// TIA Portal V17 export
// export: Created 2024-09-02T12:50:09.0439099Z, ExportSetting WithDefaults, DisplayName Totally Integrated Automation Portal, DisplayVersion V17, DisplayName TIA Portal Openness, DisplayVersion V17, DisplayName TIA Portal Version Control Interface, DisplayVersion V17, DisplayName STEP 7 Professional, DisplayVersion V17, DisplayName STEP 7 Safety, DisplayVersion V17, DisplayName WinCC Professional, DisplayVersion V17
FUNCTION_BLOCK "GraFB2_FG02_Station_OP70"   // FB1382, GRAPH
VERSION : 0.1
// stored: AcknowledgeErrorsRequired false, AutoNumber false, GraphVersion 4.0, InitialValuesAcquisition true, IsIECCheckEnabled false, LanguageInNetworks LAD, LockOperatingMode false, PermanentILProcessingInMANMode true, SetENOAutomatically false, SkipSteps false, UDAEnableTagReadback false, WithAlarmHandling true
   // inherited from GRAPH_BASE
   VAR
      OFF_SQ_BASE : Bool;
   END_VAR
   VAR_INPUT
      OFF_SQ { ExternalWritable := 'False'} : Bool := false;
      INIT_SQ { ExternalWritable := 'False'} : Bool := false;
      ACK_EF { ExternalWritable := 'False'} : Bool := false;
      S_PREV { ExternalWritable := 'False'} : Bool := false;
      S_NEXT { ExternalWritable := 'False'} : Bool := false;
      SW_AUTO { ExternalWritable := 'False'} : Bool := false;
      SW_TAP { ExternalWritable := 'False'} : Bool := false;
      SW_TOP { ExternalWritable := 'False'} : Bool := false;
      SW_MAN { ExternalWritable := 'False'} : Bool := false;
      S_SEL { ExternalWritable := 'False'} : Int := 0;
      S_ON { ExternalWritable := 'False'} : Bool := false;
      S_OFF { ExternalWritable := 'False'} : Bool := false;
      T_PUSH { ExternalWritable := 'False'} : Bool := false;
   END_VAR
   VAR_OUTPUT
      S_NO { ExternalWritable := 'False'} : Int := 0;
      S_MORE { ExternalWritable := 'False'} : Bool := false;
      S_ACTIVE { ExternalWritable := 'False'} : Bool := false;
      ERR_FLT { ExternalWritable := 'False'} : Bool := false;
      AUTO_ON { ExternalWritable := 'False'} : Bool := false;
      TAP_ON { ExternalWritable := 'False'} : Bool := false;
      TOP_ON { ExternalWritable := 'False'} : Bool := false;
      MAN_ON { ExternalWritable := 'False'} : Bool := false;
   END_VAR
   VAR
      extBlock { S7_SetPoint := 'True'} : "LTLL_ManualGraphExt";
   END_VAR
BEGIN
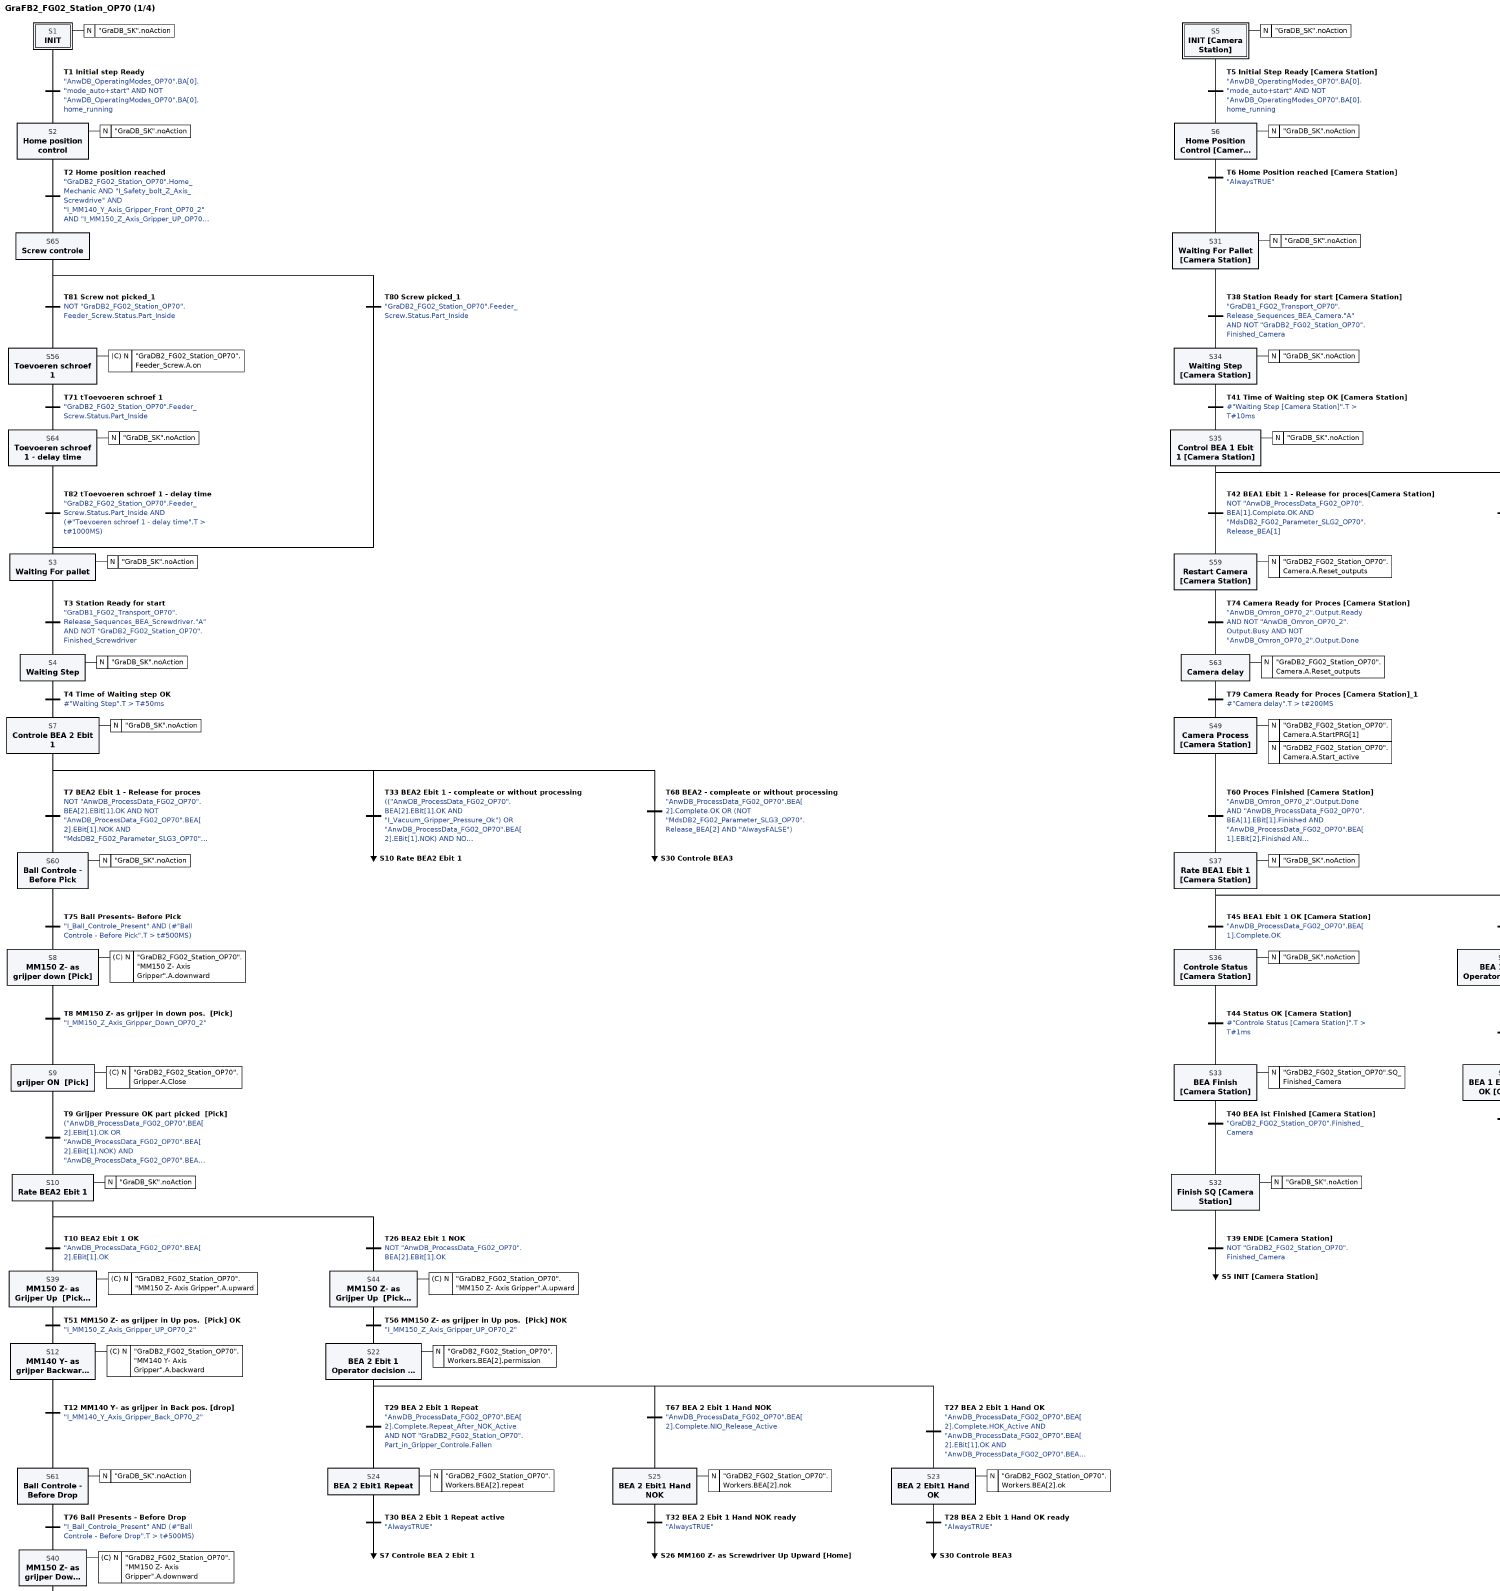
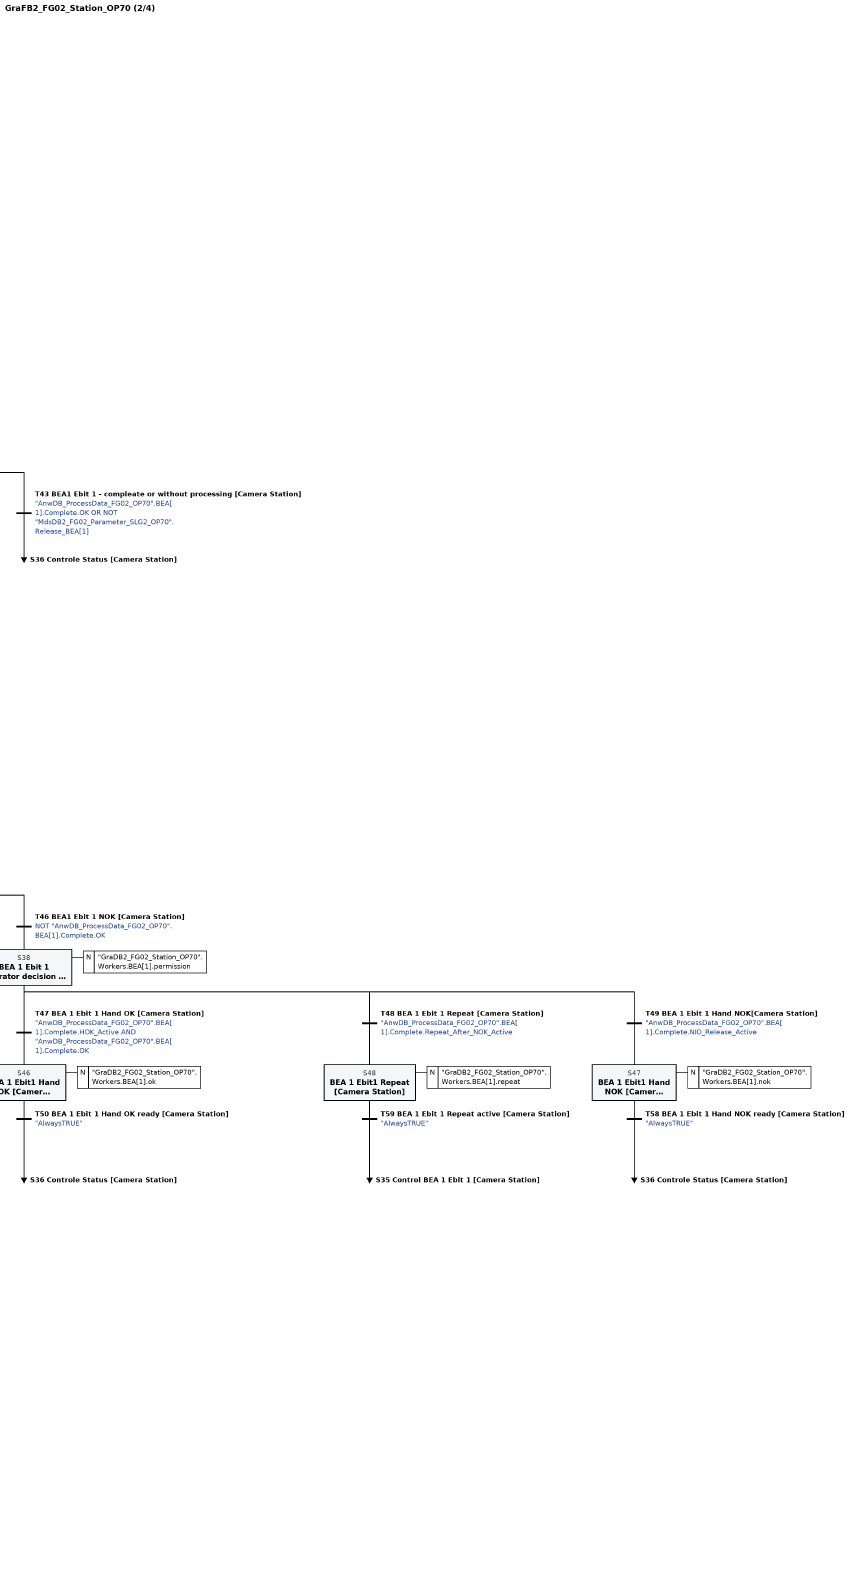
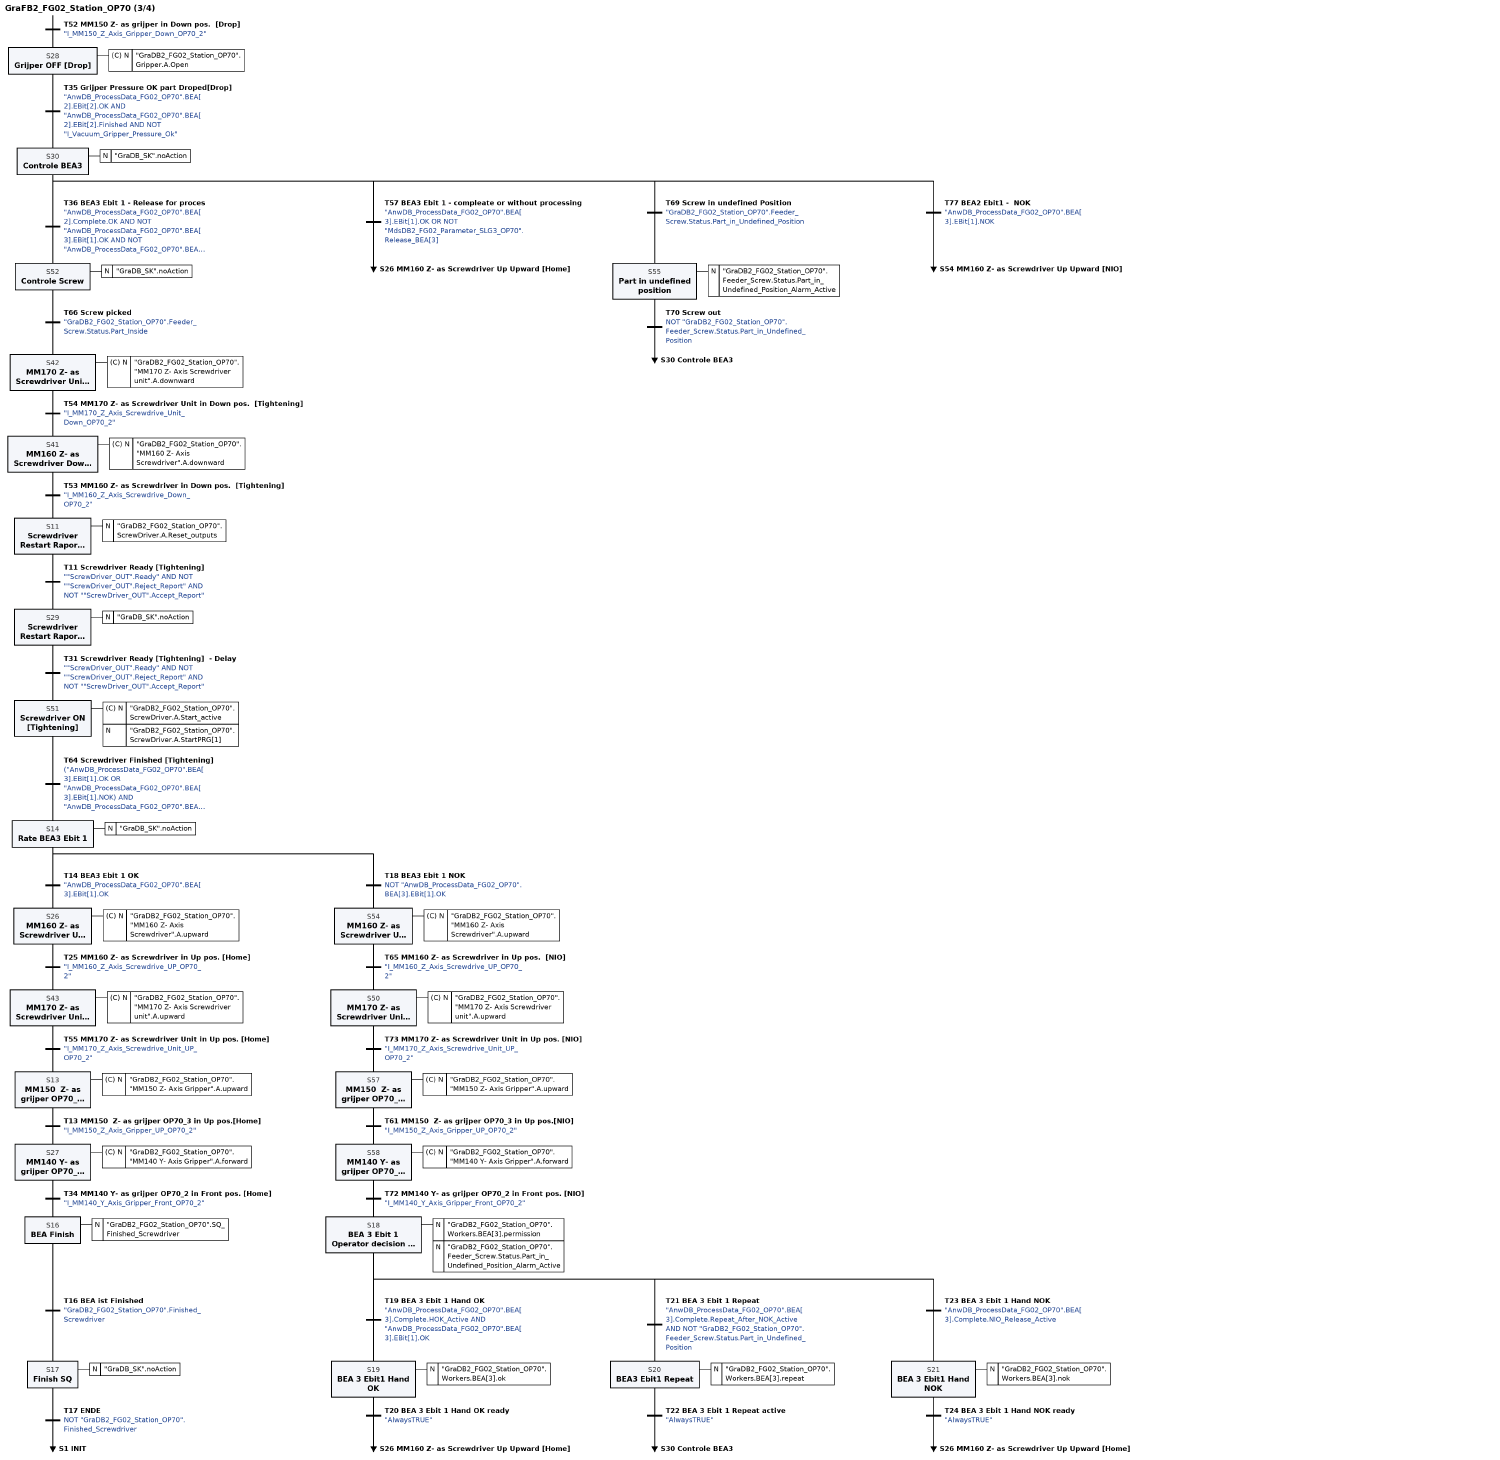
   // permanent pre-instructions
   NETWORK 1
   TITLE = HMI Lite Pass on data
      #extBlock.input := "LTLL_ManualGraphControl_OP70".screen[0].input;
   NETWORK 2
   TITLE = Instance DB Name query and pass on
      GetInstanceName(size := 0, OUT => #extBlock.input.instanceName);
   NETWORK 3
   TITLE = SK Mode
      "SysFC_SQ_Mode"(iFKT := 0, iTmsHalt := false, ioMOP := #RT_DATA.MOP);

   // sequencer 1: Station cycle Screwdriver
   // sample
   INITIAL_STEP INIT:   // S1, max time T#10S, warning time T#7S: Step commentary
      interlock C := (none);   // initial step
      supervision V := (none);   // initial step
              N    "GraDB_SK".noAction
   END_STEP
   TRANSITION "Initial step Ready" FROM INIT TO "Home position control"   // T1
      := "AnwDB_OperatingModes_OP70".BA[0]."mode_auto+start" AND NOT "AnwDB_OperatingModes_OP70".BA[0].home_running;
   END_TRANSITION
   STEP "Home position control":   // S2, max time T#10S, warning time T#7S
      supervision V := NOT #"Home position reached".TT AND (#"Home position control".U > T#1S);
      // Station
              N    "GraDB_SK".noAction
   END_STEP
   TRANSITION "Home position reached" FROM "Home position control" TO "Screw controle"   // T2
      := "GraDB2_FG02_Station_OP70".Home_Mechanic AND "I_Safety_bolt_Z_Axis_Screwdrive" AND "I_MM140_Y_Axis_Gripper_Front_OP70_2" AND "I_MM150_Z_Axis_Gripper_UP_OP70_2" AND "I_MM160_Z_Axis_Screwdrive_UP_OP70_2" AND "I_MM170_Z_Axis_Screwdrive_Unit_UP_OP70_2";
   END_TRANSITION
   STEP "Waiting For pallet":   // S3, max time T#10S, warning time T#7S
              N    "GraDB_SK".noAction
   END_STEP
   TRANSITION "Station Ready for start" FROM "Waiting For pallet" TO "Waiting Step"   // T3
      := "GraDB1_FG02_Transport_OP70".Release_Sequences_BEA_Screwdriver."A" AND NOT "GraDB2_FG02_Station_OP70".Finished_Screwdriver;
   END_TRANSITION
   STEP "Finish SQ":   // S17, max time T#10S, warning time T#7S
              N    "GraDB_SK".noAction
   END_STEP
   TRANSITION ENDE FROM "Finish SQ" TO INIT   // T17, jump
      := NOT "GraDB2_FG02_Station_OP70".Finished_Screwdriver;
   END_TRANSITION
   STEP "BEA Finish":   // S16, max time T#10S, warning time T#7S
      supervision V := NOT #"BEA ist Finished".TT AND (#"BEA Finish".U > T#1000ms);
              N    "GraDB2_FG02_Station_OP70".SQ_Finished_Screwdriver
   END_STEP
   TRANSITION "BEA ist Finished" FROM "BEA Finish" TO "Finish SQ"   // T16
      := "GraDB2_FG02_Station_OP70".Finished_Screwdriver;
   END_TRANSITION
   STEP "Waiting Step":   // S4, max time T#10S, warning time T#7S
      supervision V := NOT #"Time of Waiting step OK".TT AND (#"Waiting Step".U > t#1S);
              N    "GraDB_SK".noAction
   END_STEP
   TRANSITION "Time of Waiting step OK" FROM "Waiting Step" TO "Controle BEA 2 Ebit 1"   // T4
      := #"Waiting Step".T > T#50ms;
   END_TRANSITION
   STEP "Controle BEA 2 Ebit 1":   // S7, max time T#10S, warning time T#7S
      supervision V := NOT #"BEA2 Ebit 1 - Release for proces".TT AND (#"Controle BEA 2 Ebit 1".U > t#1s);
              N    "GraDB_SK".noAction
   END_STEP
   TRANSITION "BEA2 Ebit 1 - Release for proces" FROM "Controle BEA 2 Ebit 1" TO "Ball Controle - Before Pick"   // T7
      := NOT "AnwDB_ProcessData_FG02_OP70".BEA[2].EBit[1].OK AND NOT "AnwDB_ProcessData_FG02_OP70".BEA[2].EBit[1].NOK AND "MdsDB2_FG02_Parameter_SLG3_OP70".Release_BEA[2];
   END_TRANSITION
   TRANSITION "BEA2 Ebit 1 - compleate or without processing" FROM "Controle BEA 2 Ebit 1" TO "Rate BEA2 Ebit 1"   // T33, jump
      := (("AnwDB_ProcessData_FG02_OP70".BEA[2].EBit[1].OK AND "I_Vacuum_Gripper_Pressure_Ok") OR "AnwDB_ProcessData_FG02_OP70".BEA[2].EBit[1].NOK) AND NOT "AnwDB_ProcessData_FG02_OP70".BEA[2].EBit[2].OK;
   END_TRANSITION
   TRANSITION "BEA2 - compleate or without processing" FROM "Controle BEA 2 Ebit 1" TO "Controle BEA3"   // T68, jump
      := "AnwDB_ProcessData_FG02_OP70".BEA[2].Complete.OK OR (NOT "MdsDB2_FG02_Parameter_SLG3_OP70".Release_BEA[2] AND "AlwaysFALSE");
   END_TRANSITION
   STEP "Rate BEA2 Ebit 1":   // S10, max time T#10S, warning time T#7S: When operator access is required
      supervision V := NOT #"BEA2 Ebit 1 OK".TT AND (#"Rate BEA2 Ebit 1".U > t#1s);
              N    "GraDB_SK".noAction
   END_STEP
   TRANSITION "BEA2 Ebit 1 OK" FROM "Rate BEA2 Ebit 1" TO "MM150 Z- as Grijper Up  [Pick] OK"   // T10
      := "AnwDB_ProcessData_FG02_OP70".BEA[2].EBit[1].OK;
   END_TRANSITION
   TRANSITION "BEA2 Ebit 1 NOK" FROM "Rate BEA2 Ebit 1" TO "MM150 Z- as Grijper Up  [Pick] NOK"   // T26
      := NOT "AnwDB_ProcessData_FG02_OP70".BEA[2].EBit[1].OK;
   END_TRANSITION
   STEP "BEA 2 Ebit 1 Operator decision - After NOK":   // S22, max time T#10S, warning time T#7S
      interlock C := "GraDB1_FG02_Transport_OP70".Release_Sequences_BEA_Screwdriver."A";
              N    "GraDB2_FG02_Station_OP70".Workers.BEA[2].permission
   END_STEP
   TRANSITION "BEA 2 Ebit 1 Repeat" FROM "BEA 2 Ebit 1 Operator decision - After NOK" TO "BEA 2 Ebit1 Repeat"   // T29
      := "AnwDB_ProcessData_FG02_OP70".BEA[2].Complete.Repeat_After_NOK_Active AND NOT "GraDB2_FG02_Station_OP70".Part_in_Gripper_Controle.Fallen;
   END_TRANSITION
   TRANSITION "BEA 2 Ebit 1 Hand NOK" FROM "BEA 2 Ebit 1 Operator decision - After NOK" TO "BEA 2 Ebit1 Hand NOK"   // T67
      := "AnwDB_ProcessData_FG02_OP70".BEA[2].Complete.NIO_Release_Active;
   END_TRANSITION
   TRANSITION "BEA 2 Ebit 1 Hand OK" FROM "BEA 2 Ebit 1 Operator decision - After NOK" TO "BEA 2 Ebit1 Hand OK"   // T27
      := "AnwDB_ProcessData_FG02_OP70".BEA[2].Complete.HOK_Active AND "AnwDB_ProcessData_FG02_OP70".BEA[2].EBit[1].OK AND "AnwDB_ProcessData_FG02_OP70".BEA[2].EBit[2].OK AND NOT "GraDB2_FG02_Station_OP70".Part_in_Gripper_Controle.Fallen;
   END_TRANSITION
   STEP "BEA 2 Ebit1 Hand NOK":   // S25, max time T#10S, warning time T#7S
              N    "GraDB2_FG02_Station_OP70".Workers.BEA[2].nok
   END_STEP
   TRANSITION "BEA 2 Ebit 1 Hand NOK ready" FROM "BEA 2 Ebit1 Hand NOK" TO "MM160 Z- as Screwdriver Up Upward [Home]"   // T32, jump
      := "AlwaysTRUE";
   END_TRANSITION
   STEP "BEA 2 Ebit1 Repeat":   // S24, max time T#10S, warning time T#7S
              N    "GraDB2_FG02_Station_OP70".Workers.BEA[2].repeat
   END_STEP
   TRANSITION "BEA 2 Ebit 1 Repeat active" FROM "BEA 2 Ebit1 Repeat" TO "Controle BEA 2 Ebit 1"   // T30, jump
      := "AlwaysTRUE";
   END_TRANSITION
   STEP "MM150 Z- as Grijper Up  [Pick] OK":   // S39, max time T#10S, warning time T#7S
      interlock C := "I_MM140_Y_Axis_Gripper_Front_OP70_2" AND "I_Vacuum_Gripper_Pressure_Ok" AND NOT "AnwDB_ProcessData_FG02_OP70".BEA[2].EBit[1].NOK;
      supervision V := NOT #"MM150 Z- as grijper in Up pos.  [Pick] OK".TT AND (#"MM150 Z- as Grijper Up  [Pick] OK".U > t#1S);
      (C)     N    "GraDB2_FG02_Station_OP70"."MM150 Z- Axis Gripper".A.upward
   END_STEP
   TRANSITION "MM150 Z- as grijper in Up pos.  [Pick] OK" FROM "MM150 Z- as Grijper Up  [Pick] OK" TO "MM140 Y- as grijper Backward [drop]"   // T51
      := "I_MM150_Z_Axis_Gripper_UP_OP70_2";
   END_TRANSITION
   STEP "MM150 Z- as grijper down [Pick]":   // S8, max time T#10S, warning time T#7S
      interlock C := "I_MM70/71_index_Screwdriver_UP_OP70_2" AND "I_MM140_Y_Axis_Gripper_Front_OP70_2" AND NOT "I_Vacuum_Gripper_Pressure_Ok" AND NOT "AnwDB_ProcessData_FG02_OP70".BEA[2].EBit[1].OK;
      supervision V := NOT #"MM150 Z- as grijper in down pos.  [Pick]".TT AND (#"MM150 Z- as grijper down [Pick]".U > t#1S);
      (C)     N    "GraDB2_FG02_Station_OP70"."MM150 Z- Axis Gripper".A.downward
   END_STEP
   TRANSITION "MM150 Z- as grijper in down pos.  [Pick]" FROM "MM150 Z- as grijper down [Pick]" TO "grijper ON  [Pick]"   // T8
      := "I_MM150_Z_Axis_Gripper_Down_OP70_2";
   END_TRANSITION
   STEP "grijper ON  [Pick]":   // S9, max time T#10S, warning time T#7S
      interlock C := "I_MM70/71_index_Screwdriver_UP_OP70_2" AND "I_MM140_Y_Axis_Gripper_Front_OP70_2" AND "I_MM150_Z_Axis_Gripper_Down_OP70_2";
      supervision V := NOT #"Grijper Pressure OK part picked  [Pick]".TT AND (#"grijper ON  [Pick]".U > t#1S);
      (C)     N    "GraDB2_FG02_Station_OP70".Gripper.A.Close
   END_STEP
   TRANSITION "Grijper Pressure OK part picked  [Pick]" FROM "grijper ON  [Pick]" TO "Rate BEA2 Ebit 1"   // T9
      := ("AnwDB_ProcessData_FG02_OP70".BEA[2].EBit[1].OK OR "AnwDB_ProcessData_FG02_OP70".BEA[2].EBit[1].NOK) AND "AnwDB_ProcessData_FG02_OP70".BEA[2].EBit[1].Finished;
   END_TRANSITION
   STEP "Rate BEA3 Ebit 1":   // S14, max time T#10S, warning time T#7S: When operator access is required
      supervision V := NOT #"BEA3 Ebit 1 OK".TT AND (#"Rate BEA3 Ebit 1".U > t#1s);
              N    "GraDB_SK".noAction
   END_STEP
   TRANSITION "BEA3 Ebit 1 OK" FROM "Rate BEA3 Ebit 1" TO "MM160 Z- as Screwdriver Up Upward [Home]"   // T14
      := "AnwDB_ProcessData_FG02_OP70".BEA[3].EBit[1].OK;
   END_TRANSITION
   TRANSITION "BEA3 Ebit 1 NOK" FROM "Rate BEA3 Ebit 1" TO "MM160 Z- as Screwdriver Up Upward [NIO]"   // T18
      := NOT "AnwDB_ProcessData_FG02_OP70".BEA[3].EBit[1].OK;
   END_TRANSITION
   STEP "BEA 3 Ebit 1 Operator decision - After NOK":   // S18, max time T#10S, warning time T#7S
      interlock C := "GraDB1_FG02_Transport_OP70".Release_Sequences_BEA_Screwdriver."A";
              N    "GraDB2_FG02_Station_OP70".Workers.BEA[3].permission
              N    "GraDB2_FG02_Station_OP70".Feeder_Screw.Status.Part_in_Undefined_Position_Alarm_Active
   END_STEP
   TRANSITION "BEA 3 Ebit 1 Hand OK" FROM "BEA 3 Ebit 1 Operator decision - After NOK" TO "BEA 3 Ebit1 Hand OK"   // T19
      := "AnwDB_ProcessData_FG02_OP70".BEA[3].Complete.HOK_Active AND "AnwDB_ProcessData_FG02_OP70".BEA[3].EBit[1].OK;
   END_TRANSITION
   TRANSITION "BEA 3 Ebit 1 Repeat" FROM "BEA 3 Ebit 1 Operator decision - After NOK" TO "BEA3 Ebit1 Repeat"   // T21
      := "AnwDB_ProcessData_FG02_OP70".BEA[3].Complete.Repeat_After_NOK_Active AND NOT "GraDB2_FG02_Station_OP70".Feeder_Screw.Status.Part_in_Undefined_Position;
   END_TRANSITION
   TRANSITION "BEA 3 Ebit 1 Hand NOK" FROM "BEA 3 Ebit 1 Operator decision - After NOK" TO "BEA 3 Ebit1 Hand NOK"   // T23
      := "AnwDB_ProcessData_FG02_OP70".BEA[3].Complete.NIO_Release_Active;
   END_TRANSITION
   STEP "BEA 3 Ebit1 Hand OK":   // S19, max time T#10S, warning time T#7S
              N    "GraDB2_FG02_Station_OP70".Workers.BEA[3].ok
   END_STEP
   TRANSITION "BEA 3 Ebit 1 Hand OK ready" FROM "BEA 3 Ebit1 Hand OK" TO "MM160 Z- as Screwdriver Up Upward [Home]"   // T20, jump
      := "AlwaysTRUE";
   END_TRANSITION
   STEP "BEA 3 Ebit1 Hand NOK":   // S21, max time T#10S, warning time T#7S
              N    "GraDB2_FG02_Station_OP70".Workers.BEA[3].nok
   END_STEP
   TRANSITION "BEA 3 Ebit 1 Hand NOK ready" FROM "BEA 3 Ebit1 Hand NOK" TO "MM160 Z- as Screwdriver Up Upward [Home]"   // T24, jump
      := "AlwaysTRUE";
   END_TRANSITION
   STEP "BEA3 Ebit1 Repeat":   // S20, max time T#10S, warning time T#7S
              N    "GraDB2_FG02_Station_OP70".Workers.BEA[3].repeat
   END_STEP
   TRANSITION "BEA 3 Ebit 1 Repeat active" FROM "BEA3 Ebit1 Repeat" TO "Controle BEA3"   // T22, jump
      := "AlwaysTRUE";
   END_TRANSITION
   STEP "MM150 Z- as grijper Down [Drop]":   // S40, max time T#10S, warning time T#7S
      interlock C := "I_MM70/71_index_Screwdriver_UP_OP70_2" AND "I_MM140_Y_Axis_Gripper_Back_OP70_2" AND "I_Vacuum_Gripper_Pressure_Ok" AND "AnwDB_ProcessData_FG02_OP70".BEA[2].EBit[1].OK AND NOT "AnwDB_ProcessData_FG02_OP70".BEA[2].EBit[1].NOK;
      supervision V := NOT #"MM150 Z- as grijper in Down pos.  [Drop]".TT AND (#"MM150 Z- as grijper Down [Drop]".U > t#1S);
      (C)     N    "GraDB2_FG02_Station_OP70"."MM150 Z- Axis Gripper".A.downward
   END_STEP
   TRANSITION "MM150 Z- as grijper in Down pos.  [Drop]" FROM "MM150 Z- as grijper Down [Drop]" TO "Grijper OFF [Drop]"   // T52
      := "I_MM150_Z_Axis_Gripper_Down_OP70_2";
   END_TRANSITION
   STEP "Screwdriver Restart Raport [Tightening]":   // S11, max time T#10S, warning time T#7S
      interlock C := "AlwaysTRUE";
      supervision V := NOT #"Screwdriver Ready [Tightening]".TT AND (#"Screwdriver Restart Raport [Tightening]".U > t#10S);
              N    "GraDB2_FG02_Station_OP70".ScrewDriver.A.Reset_outputs
   END_STEP
   TRANSITION "Screwdriver Ready [Tightening]" FROM "Screwdriver Restart Raport [Tightening]" TO "Screwdriver Restart Raport [Tightening] - Delay"   // T11
      := ""ScrewDriver_OUT".Ready" AND NOT ""ScrewDriver_OUT".Reject_Report" AND NOT ""ScrewDriver_OUT".Accept_Report";
   END_TRANSITION
   STEP "MM160 Z- as Screwdriver Up Upward [Home]":   // S26, max time T#10S, warning time T#7S
      interlock C := "AlwaysTRUE";
      supervision V := NOT #"MM160 Z- as Screwdriver in Up pos. [Home]".TT AND (#"MM160 Z- as Screwdriver Up Upward [Home]".U > T#5S);
      (C)     N    "GraDB2_FG02_Station_OP70"."MM160 Z- Axis Screwdriver".A.upward
   END_STEP
   TRANSITION "MM160 Z- as Screwdriver in Up pos. [Home]" FROM "MM160 Z- as Screwdriver Up Upward [Home]" TO "MM170 Z- as Screwdriver Unit Up [Home]"   // T25
      := "I_MM160_Z_Axis_Screwdrive_UP_OP70_2";
   END_TRANSITION
   STEP "MM160 Z- as Screwdriver Down [Tightening]":   // S41, max time T#10S, warning time T#7S
      interlock C := "I_MM70/71_index_Screwdriver_UP_OP70_2" AND "I_MM170_Z_Axis_Screwdrive_Unit_Down_OP70_2" AND (("I_MM140_Y_Axis_Gripper_Back_OP70_2" AND "I_MM150_Z_Axis_Gripper_Down_OP70_2") OR ("I_MM140_Y_Axis_Gripper_Front_OP70_2" AND "I_MM150_Z_Axis_Gripper_UP_OP70_2")) AND "AnwDB_ProcessData_FG02_OP70".BEA[2].Complete.OK;
      supervision V := NOT #"MM160 Z- as Screwdriver in Down pos.  [Tightening]".TT AND (#"MM160 Z- as Screwdriver Down [Tightening]".U > t#1S);
      (C)     N    "GraDB2_FG02_Station_OP70"."MM160 Z- Axis Screwdriver".A.downward
   END_STEP
   TRANSITION "MM160 Z- as Screwdriver in Down pos.  [Tightening]" FROM "MM160 Z- as Screwdriver Down [Tightening]" TO "Screwdriver Restart Raport [Tightening]"   // T53
      := "I_MM160_Z_Axis_Screwdrive_Down_OP70_2";
   END_TRANSITION
   STEP "MM170 Z- as Screwdriver Unit Down [Tightening]":   // S42, max time T#10S, warning time T#7S
      interlock C := "I_MM70/71_index_Screwdriver_UP_OP70_2" AND "I_MM160_Z_Axis_Screwdrive_UP_OP70_2" AND (("I_MM140_Y_Axis_Gripper_Back_OP70_2" AND "I_MM150_Z_Axis_Gripper_Down_OP70_2") OR ("I_MM140_Y_Axis_Gripper_Front_OP70_2" AND "I_MM150_Z_Axis_Gripper_UP_OP70_2")) AND "I_Safety_bolt_Z_Axis_Screwdrive" AND "AnwDB_ProcessData_FG02_OP70".BEA[2].Complete.OK;
      supervision V := NOT #"MM170 Z- as Screwdriver Unit in Down pos.  [Tightening]".TT AND (#"MM170 Z- as Screwdriver Unit Down [Tightening]".U > t#1S);
      (C)     N    "GraDB2_FG02_Station_OP70"."MM170 Z- Axis Screwdriver unit".A.downward
   END_STEP
   TRANSITION "MM170 Z- as Screwdriver Unit in Down pos.  [Tightening]" FROM "MM170 Z- as Screwdriver Unit Down [Tightening]" TO "MM160 Z- as Screwdriver Down [Tightening]"   // T54
      := "I_MM170_Z_Axis_Screwdrive_Unit_Down_OP70_2";
   END_TRANSITION
   STEP "MM170 Z- as Screwdriver Unit Up [Home]":   // S43, max time T#10S, warning time T#7S
      interlock C := "I_MM160_Z_Axis_Screwdrive_UP_OP70_2" AND (("I_MM140_Y_Axis_Gripper_Back_OP70_2" AND "I_MM150_Z_Axis_Gripper_Down_OP70_2") OR ("I_MM140_Y_Axis_Gripper_Front_OP70_2" AND "I_MM150_Z_Axis_Gripper_UP_OP70_2")) AND "I_Safety_bolt_Z_Axis_Screwdrive";
      supervision V := NOT #"MM170 Z- as Screwdriver Unit in Up pos. [Home]".TT AND (#"MM170 Z- as Screwdriver Unit Up [Home]".U > t#1S);
      (C)     N    "GraDB2_FG02_Station_OP70"."MM170 Z- Axis Screwdriver unit".A.upward
   END_STEP
   TRANSITION "MM170 Z- as Screwdriver Unit in Up pos. [Home]" FROM "MM170 Z- as Screwdriver Unit Up [Home]" TO "MM150  Z- as grijper OP70_3 Upward [Home]"   // T55
      := "I_MM170_Z_Axis_Screwdrive_Unit_UP_OP70_2";
   END_TRANSITION
   STEP "MM150  Z- as grijper OP70_3 Upward [Home]":   // S13, max time T#10S, warning time T#7S
      interlock C := "I_MM160_Z_Axis_Screwdrive_UP_OP70_2" AND "I_MM170_Z_Axis_Screwdrive_Unit_UP_OP70_2" AND (NOT "AnwDB_ProcessData_FG02_OP70".BEA[3].Complete.OK OR ("AnwDB_ProcessData_FG02_OP70".BEA[3].Complete.OK AND NOT "I_Vacuum_Gripper_Pressure_Ok"));
      supervision V := NOT #"MM150  Z- as grijper OP70_3 in Up pos.[Home]".TT AND (#"MM150  Z- as grijper OP70_3 Upward [Home]".U > T#5S);
      (C)     N    "GraDB2_FG02_Station_OP70"."MM150 Z- Axis Gripper".A.upward
   END_STEP
   TRANSITION "MM150  Z- as grijper OP70_3 in Up pos.[Home]" FROM "MM150  Z- as grijper OP70_3 Upward [Home]" TO "MM140 Y- as grijper OP70_2 Forward[Home]"   // T13
      := "I_MM150_Z_Axis_Gripper_UP_OP70_2";
   END_TRANSITION
   STEP "MM150 Z- as Grijper Up  [Pick] NOK":   // S44, max time T#10S, warning time T#7S
      interlock C := "I_MM140_Y_Axis_Gripper_Front_OP70_2";
      supervision V := NOT #"MM150 Z- as grijper in Up pos.  [Pick] NOK".TT AND (#"MM150 Z- as Grijper Up  [Pick] NOK".U > t#1S);
      (C)     N    "GraDB2_FG02_Station_OP70"."MM150 Z- Axis Gripper".A.upward
   END_STEP
   TRANSITION "MM150 Z- as grijper in Up pos.  [Pick] NOK" FROM "MM150 Z- as Grijper Up  [Pick] NOK" TO "BEA 2 Ebit 1 Operator decision - After NOK"   // T56
      := "I_MM150_Z_Axis_Gripper_UP_OP70_2";
   END_TRANSITION
   STEP "MM140 Y- as grijper Backward [drop]":   // S12, max time T#10S, warning time T#7S
      interlock C := "I_MM150_Z_Axis_Gripper_UP_OP70_2" AND "I_MM160_Z_Axis_Screwdrive_UP_OP70_2" AND "I_MM170_Z_Axis_Screwdrive_Unit_UP_OP70_2" AND "I_Vacuum_Gripper_Pressure_Ok" AND "AnwDB_ProcessData_FG02_OP70".BEA[2].EBit[1].OK AND NOT "AnwDB_ProcessData_FG02_OP70".BEA[2].EBit[1].NOK;
      supervision V := NOT #"MM140 Y- as grijper in Back pos. [drop]".TT AND (#"MM140 Y- as grijper Backward [drop]".U > t#1S);
      (C)     N    "GraDB2_FG02_Station_OP70"."MM140 Y- Axis Gripper".A.backward
   END_STEP
   TRANSITION "MM140 Y- as grijper in Back pos. [drop]" FROM "MM140 Y- as grijper Backward [drop]" TO "Ball Controle - Before Drop"   // T12
      := "I_MM140_Y_Axis_Gripper_Back_OP70_2";
   END_TRANSITION
   STEP "MM140 Y- as grijper OP70_2 Forward[Home]":   // S27, max time T#10S, warning time T#7S
      interlock C := "I_MM150_Z_Axis_Gripper_UP_OP70_2" AND "I_MM160_Z_Axis_Screwdrive_UP_OP70_2" AND "I_MM170_Z_Axis_Screwdrive_Unit_UP_OP70_2";
      supervision V := NOT #"MM140 Y- as grijper OP70_2 in Front pos. [Home]".TT AND (#"MM140 Y- as grijper OP70_2 Forward[Home]".U > T#5S);
      (C)     N    "GraDB2_FG02_Station_OP70"."MM140 Y- Axis Gripper".A.forward
   END_STEP
   TRANSITION "MM140 Y- as grijper OP70_2 in Front pos. [Home]" FROM "MM140 Y- as grijper OP70_2 Forward[Home]" TO "BEA Finish"   // T34
      := "I_MM140_Y_Axis_Gripper_Front_OP70_2";
   END_TRANSITION
   STEP "Grijper OFF [Drop]":   // S28, max time T#10S, warning time T#7S
      interlock C := "I_MM70/71_index_Screwdriver_UP_OP70_2" AND "I_MM140_Y_Axis_Gripper_Back_OP70_2" AND "I_MM150_Z_Axis_Gripper_Down_OP70_2";
      supervision V := NOT #"Grijper Pressure OK part Droped[Drop]".TT AND (#"Grijper OFF [Drop]".U > t#1S);
      (C)     N    "GraDB2_FG02_Station_OP70".Gripper.A.Open
   END_STEP
   TRANSITION "Grijper Pressure OK part Droped[Drop]" FROM "Grijper OFF [Drop]" TO "Controle BEA3"   // T35
      := "AnwDB_ProcessData_FG02_OP70".BEA[2].EBit[2].OK AND "AnwDB_ProcessData_FG02_OP70".BEA[2].EBit[2].Finished AND NOT "I_Vacuum_Gripper_Pressure_Ok";
   END_TRANSITION
   STEP "Controle Screw":   // S52, max time T#10S, warning time T#7S
      supervision V := #"Controle Screw".U > t#1S;
              N    "GraDB_SK".noAction
   END_STEP
   TRANSITION "Screw picked" FROM "Controle Screw" TO "MM170 Z- as Screwdriver Unit Down [Tightening]"   // T66
      := "GraDB2_FG02_Station_OP70".Feeder_Screw.Status.Part_Inside;
   END_TRANSITION
   STEP "Screwdriver ON  [Tightening]":   // S51, max time T#10S, warning time T#7S
      interlock C := "I_MM70/71_index_Screwdriver_UP_OP70_2" AND (("I_MM140_Y_Axis_Gripper_Back_OP70_2" AND "I_MM150_Z_Axis_Gripper_Down_OP70_2") OR ("I_MM140_Y_Axis_Gripper_Front_OP70_2" AND "I_MM150_Z_Axis_Gripper_UP_OP70_2")) AND "I_MM160_Z_Axis_Screwdrive_Down_OP70_2" AND "I_MM170_Z_Axis_Screwdrive_Unit_Down_OP70_2" AND "AnwDB_ProcessData_FG02_OP70".BEA[2].Complete.OK;
      supervision V := NOT #"Screwdriver Finished [Tightening]".TT AND (#"Screwdriver ON  [Tightening]".U > t#10S);
      (C)     N    "GraDB2_FG02_Station_OP70".ScrewDriver.A.Start_active
              N    "GraDB2_FG02_Station_OP70".ScrewDriver.A.StartPRG[1]
   END_STEP
   TRANSITION "Screwdriver Finished [Tightening]" FROM "Screwdriver ON  [Tightening]" TO "Rate BEA3 Ebit 1"   // T64
      := ("AnwDB_ProcessData_FG02_OP70".BEA[3].EBit[1].OK OR "AnwDB_ProcessData_FG02_OP70".BEA[3].EBit[1].NOK) AND "AnwDB_ProcessData_FG02_OP70".BEA[3].EBit[1].Finished;
   END_TRANSITION
   STEP "MM160 Z- as Screwdriver Up Upward [NIO]":   // S54, max time T#10S, warning time T#7S
      interlock C := "AlwaysTRUE";
      supervision V := NOT #"MM160 Z- as Screwdriver in Up pos.  [NIO]".TT AND (#"MM160 Z- as Screwdriver Up Upward [NIO]".U > T#5S);
      (C)     N    "GraDB2_FG02_Station_OP70"."MM160 Z- Axis Screwdriver".A.upward
   END_STEP
   TRANSITION "MM160 Z- as Screwdriver in Up pos.  [NIO]" FROM "MM160 Z- as Screwdriver Up Upward [NIO]" TO "MM170 Z- as Screwdriver Unit Up [NIO]"   // T65
      := "I_MM160_Z_Axis_Screwdrive_UP_OP70_2";
   END_TRANSITION
   STEP "BEA 2 Ebit1 Hand OK":   // S23, max time T#10S, warning time T#7S
              N    "GraDB2_FG02_Station_OP70".Workers.BEA[2].ok
   END_STEP
   TRANSITION "BEA 2 Ebit 1 Hand OK ready" FROM "BEA 2 Ebit1 Hand OK" TO "Controle BEA3"   // T28, jump
      := "AlwaysTRUE";
   END_TRANSITION
   STEP "Controle BEA3":   // S30, max time T#10S, warning time T#7S
      supervision V := NOT #"BEA3 Ebit 1 - Release for proces".TT AND (#"Controle BEA3".U > t#1s);
              N    "GraDB_SK".noAction
   END_STEP
   TRANSITION "BEA3 Ebit 1 - Release for proces" FROM "Controle BEA3" TO "Controle Screw"   // T36
      := "AnwDB_ProcessData_FG02_OP70".BEA[2].Complete.OK AND NOT "AnwDB_ProcessData_FG02_OP70".BEA[3].EBit[1].OK AND NOT "AnwDB_ProcessData_FG02_OP70".BEA[3].EBit[1].NOK AND NOT "GraDB2_FG02_Station_OP70".Feeder_Screw.Status.Part_in_Undefined_Position AND "MdsDB2_FG02_Parameter_SLG3_OP70".Release_BEA[3];
   END_TRANSITION
   TRANSITION "BEA3 Ebit 1 - compleate or without processing" FROM "Controle BEA3" TO "MM160 Z- as Screwdriver Up Upward [Home]"   // T57, jump
      := "AnwDB_ProcessData_FG02_OP70".BEA[3].EBit[1].OK OR NOT "MdsDB2_FG02_Parameter_SLG3_OP70".Release_BEA[3];
   END_TRANSITION
   TRANSITION "Screw in undefined Position" FROM "Controle BEA3" TO "Part in undefined position"   // T69
      := "GraDB2_FG02_Station_OP70".Feeder_Screw.Status.Part_in_Undefined_Position;
   END_TRANSITION
   TRANSITION "BEA2 Ebit1 -  NOK" FROM "Controle BEA3" TO "MM160 Z- as Screwdriver Up Upward [NIO]"   // T77, jump
      := "AnwDB_ProcessData_FG02_OP70".BEA[3].EBit[1].NOK;
   END_TRANSITION
   STEP "Part in undefined position":   // S55, max time T#10S, warning time T#7S
      supervision V := NOT #"Screw out".TT AND (#"Part in undefined position".U > t#7S);
              N    "GraDB2_FG02_Station_OP70".Feeder_Screw.Status.Part_in_Undefined_Position_Alarm_Active
   END_STEP
   TRANSITION "Screw out" FROM "Part in undefined position" TO "Controle BEA3"   // T70, jump
      := NOT "GraDB2_FG02_Station_OP70".Feeder_Screw.Status.Part_in_Undefined_Position;
   END_TRANSITION
   STEP "MM170 Z- as Screwdriver Unit Up [NIO]":   // S50, max time T#10S, warning time T#7S
      interlock C := "I_MM160_Z_Axis_Screwdrive_UP_OP70_2" AND (("I_MM140_Y_Axis_Gripper_Back_OP70_2" AND "I_MM150_Z_Axis_Gripper_Down_OP70_2") OR ("I_MM140_Y_Axis_Gripper_Front_OP70_2" AND "I_MM150_Z_Axis_Gripper_UP_OP70_2")) AND "I_Safety_bolt_Z_Axis_Screwdrive";
      supervision V := NOT #"MM170 Z- as Screwdriver Unit in Up pos. [NIO]".TT AND (#"MM170 Z- as Screwdriver Unit Up [NIO]".U > t#1S);
      (C)     N    "GraDB2_FG02_Station_OP70"."MM170 Z- Axis Screwdriver unit".A.upward
   END_STEP
   TRANSITION "MM170 Z- as Screwdriver Unit in Up pos. [NIO]" FROM "MM170 Z- as Screwdriver Unit Up [NIO]" TO "MM150  Z- as grijper OP70_3 Upward [NIO]"   // T73
      := "I_MM170_Z_Axis_Screwdrive_Unit_UP_OP70_2";
   END_TRANSITION
   STEP "MM150  Z- as grijper OP70_3 Upward [NIO]":   // S57, max time T#10S, warning time T#7S
      interlock C := "I_MM160_Z_Axis_Screwdrive_UP_OP70_2" AND "I_MM170_Z_Axis_Screwdrive_Unit_UP_OP70_2" AND (NOT "AnwDB_ProcessData_FG02_OP70".BEA[3].Complete.OK OR ("AnwDB_ProcessData_FG02_OP70".BEA[3].Complete.OK AND NOT "I_Vacuum_Gripper_Pressure_Ok"));
      supervision V := NOT #"MM150  Z- as grijper OP70_3 in Up pos.[NIO]".TT AND (#"MM150  Z- as grijper OP70_3 Upward [NIO]".U > T#5S);
      (C)     N    "GraDB2_FG02_Station_OP70"."MM150 Z- Axis Gripper".A.upward
   END_STEP
   TRANSITION "MM150  Z- as grijper OP70_3 in Up pos.[NIO]" FROM "MM150  Z- as grijper OP70_3 Upward [NIO]" TO "MM140 Y- as grijper OP70_2 Forward [NIO]"   // T61
      := "I_MM150_Z_Axis_Gripper_UP_OP70_2";
   END_TRANSITION
   STEP "MM140 Y- as grijper OP70_2 Forward [NIO]":   // S58, max time T#10S, warning time T#7S
      interlock C := "I_MM150_Z_Axis_Gripper_UP_OP70_2" AND "I_MM160_Z_Axis_Screwdrive_UP_OP70_2" AND "I_MM170_Z_Axis_Screwdrive_Unit_UP_OP70_2";
      supervision V := NOT #"MM140 Y- as grijper OP70_2 in Front pos. [NIO]".TT AND (#"MM140 Y- as grijper OP70_2 Forward [NIO]".U > T#5S);
      (C)     N    "GraDB2_FG02_Station_OP70"."MM140 Y- Axis Gripper".A.forward
   END_STEP
   TRANSITION "MM140 Y- as grijper OP70_2 in Front pos. [NIO]" FROM "MM140 Y- as grijper OP70_2 Forward [NIO]" TO "BEA 3 Ebit 1 Operator decision - After NOK"   // T72
      := "I_MM140_Y_Axis_Gripper_Front_OP70_2";
   END_TRANSITION
   STEP "Ball Controle - Before Pick":   // S60, max time T#10S, warning time T#7S
      supervision V := NOT #"Ball Presents- Before Pick".TT AND (#"Ball Controle - Before Pick".U > t#1S);
              N    "GraDB_SK".noAction
   END_STEP
   TRANSITION "Ball Presents- Before Pick" FROM "Ball Controle - Before Pick" TO "MM150 Z- as grijper down [Pick]"   // T75
      := "I_Ball_Controle_Present" AND (#"Ball Controle - Before Pick".T > t#500MS);
   END_TRANSITION
   STEP "Ball Controle - Before Drop":   // S61, max time T#10S, warning time T#7S
      supervision V := NOT #"Ball Presents - Before Drop".TT AND (#"Ball Controle - Before Drop".U > t#1S);
              N    "GraDB_SK".noAction
   END_STEP
   TRANSITION "Ball Presents - Before Drop" FROM "Ball Controle - Before Drop" TO "MM150 Z- as grijper Down [Drop]"   // T76
      := "I_Ball_Controle_Present" AND (#"Ball Controle - Before Drop".T > t#500MS);
   END_TRANSITION
   STEP "Screwdriver Restart Raport [Tightening] - Delay":   // S29, max time T#10S, warning time T#7S
      interlock C := "AlwaysTRUE";
      supervision V := NOT #"Screwdriver Ready [Tightening]  - Delay".TT AND (#"Screwdriver Restart Raport [Tightening] - Delay".U > t#10S);
              N    "GraDB_SK".noAction
   END_STEP
   TRANSITION "Screwdriver Ready [Tightening]  - Delay" FROM "Screwdriver Restart Raport [Tightening] - Delay" TO "Screwdriver ON  [Tightening]"   // T31
      := ""ScrewDriver_OUT".Ready" AND NOT ""ScrewDriver_OUT".Reject_Report" AND NOT ""ScrewDriver_OUT".Accept_Report";
   END_TRANSITION
   STEP "Screw controle":   // S65, max time T#10S, warning time T#7S
   END_STEP
   TRANSITION "Screw not picked_1" FROM "Screw controle" TO "Toevoeren schroef 1"   // T81
      := NOT "GraDB2_FG02_Station_OP70".Feeder_Screw.Status.Part_Inside;
   END_TRANSITION
   TRANSITION "Screw picked_1" FROM "Screw controle" TO "Waiting For pallet"   // T80
      := "GraDB2_FG02_Station_OP70".Feeder_Screw.Status.Part_Inside;
   END_TRANSITION
   STEP "Toevoeren schroef 1":   // S56, max time T#10S, warning time T#7S
      supervision V := NOT #"tToevoeren schroef 1".TT AND (#"Toevoeren schroef 1".U > t#7S);
      (C)     N    "GraDB2_FG02_Station_OP70".Feeder_Screw.A.on
   END_STEP
   TRANSITION "tToevoeren schroef 1" FROM "Toevoeren schroef 1" TO "Toevoeren schroef 1 - delay time"   // T71
      := "GraDB2_FG02_Station_OP70".Feeder_Screw.Status.Part_Inside;
   END_TRANSITION
   STEP "Toevoeren schroef 1 - delay time":   // S64, max time T#10S, warning time T#7S
      supervision V := NOT #"tToevoeren schroef 1 - delay time".TT AND (#"Toevoeren schroef 1 - delay time".U > t#7S);
              N    "GraDB_SK".noAction
   END_STEP
   TRANSITION "tToevoeren schroef 1 - delay time" FROM "Toevoeren schroef 1 - delay time" TO "Waiting For pallet"   // T82
      := "GraDB2_FG02_Station_OP70".Feeder_Screw.Status.Part_Inside AND (#"Toevoeren schroef 1 - delay time".T > t#1000MS);
   END_TRANSITION

   // sequencer 2: Station Cycle Camera
   INITIAL_STEP "INIT [Camera Station]":   // S5, max time T#10S, warning time T#7S: Step commentary
      interlock C := (none);   // initial step
      supervision V := (none);   // initial step
              N    "GraDB_SK".noAction
   END_STEP
   TRANSITION "Initial Step Ready [Camera Station]" FROM "INIT [Camera Station]" TO "Home Position Control [Camera Station]"   // T5
      := "AnwDB_OperatingModes_OP70".BA[0]."mode_auto+start" AND NOT "AnwDB_OperatingModes_OP70".BA[0].home_running;
   END_TRANSITION
   STEP "Home Position Control [Camera Station]":   // S6, max time T#10S, warning time T#7S
      supervision V := NOT #"Home Position reached [Camera Station]".TT AND (#"Home Position Control [Camera Station]".U > T#1S);
      // Station
              N    "GraDB_SK".noAction
   END_STEP
   TRANSITION "Home Position reached [Camera Station]" FROM "Home Position Control [Camera Station]" TO "Waiting For Pallet [Camera Station]"   // T6
      := "AlwaysTRUE";
   END_TRANSITION
   STEP "Waiting For Pallet [Camera Station]":   // S31, max time T#10S, warning time T#7S
              N    "GraDB_SK".noAction
   END_STEP
   TRANSITION "Station Ready for start [Camera Station]" FROM "Waiting For Pallet [Camera Station]" TO "Waiting Step [Camera Station]"   // T38
      := "GraDB1_FG02_Transport_OP70".Release_Sequences_BEA_Camera."A" AND NOT "GraDB2_FG02_Station_OP70".Finished_Camera;
   END_TRANSITION
   STEP "Finish SQ [Camera Station]":   // S32, max time T#10S, warning time T#7S
              N    "GraDB_SK".noAction
   END_STEP
   TRANSITION "ENDE [Camera Station]" FROM "Finish SQ [Camera Station]" TO "INIT [Camera Station]"   // T39, jump
      := NOT "GraDB2_FG02_Station_OP70".Finished_Camera;
   END_TRANSITION
   STEP "BEA Finish [Camera Station]":   // S33, max time T#10S, warning time T#7S
      supervision V := NOT #"BEA ist Finished [Camera Station]".TT AND (#"BEA Finish [Camera Station]".U > T#1000ms);
              N    "GraDB2_FG02_Station_OP70".SQ_Finished_Camera
   END_STEP
   TRANSITION "BEA ist Finished [Camera Station]" FROM "BEA Finish [Camera Station]" TO "Finish SQ [Camera Station]"   // T40
      := "GraDB2_FG02_Station_OP70".Finished_Camera;
   END_TRANSITION
   STEP "Waiting Step [Camera Station]":   // S34, max time T#10S, warning time T#7S
      supervision V := NOT #"Time of Waiting step OK [Camera Station]".TT AND (#"Waiting Step [Camera Station]".U > t#1S);
              N    "GraDB_SK".noAction
   END_STEP
   TRANSITION "Time of Waiting step OK [Camera Station]" FROM "Waiting Step [Camera Station]" TO "Control BEA 1 Ebit 1 [Camera Station]"   // T41
      := #"Waiting Step [Camera Station]".T > T#10ms;
   END_TRANSITION
   STEP "Control BEA 1 Ebit 1 [Camera Station]":   // S35, max time T#10S, warning time T#7S
      supervision V := NOT #"BEA1 Ebit 1 - Release for proces[Camera Station]".TT AND (#"Control BEA 1 Ebit 1 [Camera Station]".U > t#1s);
              N    "GraDB_SK".noAction
   END_STEP
   TRANSITION "BEA1 Ebit 1 - Release for proces[Camera Station]" FROM "Control BEA 1 Ebit 1 [Camera Station]" TO "Restart Camera  [Camera Station]"   // T42
      := NOT "AnwDB_ProcessData_FG02_OP70".BEA[1].Complete.OK AND "MdsDB2_FG02_Parameter_SLG2_OP70".Release_BEA[1];
   END_TRANSITION
   TRANSITION "BEA1 Ebit 1 - compleate or without processing [Camera Station]" FROM "Control BEA 1 Ebit 1 [Camera Station]" TO "Controle Status [Camera Station]"   // T43, jump
      := "AnwDB_ProcessData_FG02_OP70".BEA[1].Complete.OK OR NOT "MdsDB2_FG02_Parameter_SLG2_OP70".Release_BEA[1];
   END_TRANSITION
   STEP "Controle Status [Camera Station]":   // S36, max time T#10S, warning time T#7S
      supervision V := NOT #"Status OK [Camera Station]".TT AND (#"Controle Status [Camera Station]".U > T#5s);
              N    "GraDB_SK".noAction
   END_STEP
   TRANSITION "Status OK [Camera Station]" FROM "Controle Status [Camera Station]" TO "BEA Finish [Camera Station]"   // T44
      := #"Controle Status [Camera Station]".T > T#1ms;
   END_TRANSITION
   STEP "Rate BEA1 Ebit 1 [Camera Station]":   // S37, max time T#10S, warning time T#7S: When operator access is required
      supervision V := NOT #"BEA1 Ebit 1 OK [Camera Station]".TT AND (#"Rate BEA1 Ebit 1 [Camera Station]".U > t#1s);
              N    "GraDB_SK".noAction
   END_STEP
   TRANSITION "BEA1 Ebit 1 OK [Camera Station]" FROM "Rate BEA1 Ebit 1 [Camera Station]" TO "Controle Status [Camera Station]"   // T45
      := "AnwDB_ProcessData_FG02_OP70".BEA[1].Complete.OK;
   END_TRANSITION
   TRANSITION "BEA1 Ebit 1 NOK [Camera Station]" FROM "Rate BEA1 Ebit 1 [Camera Station]" TO "BEA 1 Ebit 1 Operator decision - After NOK [Camera Station]"   // T46
      := NOT "AnwDB_ProcessData_FG02_OP70".BEA[1].Complete.OK;
   END_TRANSITION
   STEP "BEA 1 Ebit 1 Operator decision - After NOK [Camera Station]":   // S38, max time T#10S, warning time T#7S
      interlock C := "GraDB1_FG02_Transport_OP70".Release_Sequences_BEA_Camera."A";
              N    "GraDB2_FG02_Station_OP70".Workers.BEA[1].permission
   END_STEP
   TRANSITION "BEA 1 Ebit 1 Hand OK [Camera Station]" FROM "BEA 1 Ebit 1 Operator decision - After NOK [Camera Station]" TO "BEA 1 Ebit1 Hand OK [Camera Station]"   // T47
      := "AnwDB_ProcessData_FG02_OP70".BEA[1].Complete.HOK_Active AND "AnwDB_ProcessData_FG02_OP70".BEA[1].Complete.OK;
   END_TRANSITION
   TRANSITION "BEA 1 Ebit 1 Repeat [Camera Station]" FROM "BEA 1 Ebit 1 Operator decision - After NOK [Camera Station]" TO "BEA 1 Ebit1 Repeat [Camera Station]"   // T48
      := "AnwDB_ProcessData_FG02_OP70".BEA[1].Complete.Repeat_After_NOK_Active;
   END_TRANSITION
   TRANSITION "BEA 1 Ebit 1 Hand NOK[Camera Station]" FROM "BEA 1 Ebit 1 Operator decision - After NOK [Camera Station]" TO "BEA 1 Ebit1 Hand NOK [Camera Station]"   // T49
      := "AnwDB_ProcessData_FG02_OP70".BEA[1].Complete.NIO_Release_Active;
   END_TRANSITION
   STEP "BEA 1 Ebit1 Hand OK [Camera Station]":   // S46, max time T#10S, warning time T#7S
              N    "GraDB2_FG02_Station_OP70".Workers.BEA[1].ok
   END_STEP
   TRANSITION "BEA 1 Ebit 1 Hand OK ready [Camera Station]" FROM "BEA 1 Ebit1 Hand OK [Camera Station]" TO "Controle Status [Camera Station]"   // T50, jump
      := "AlwaysTRUE";
   END_TRANSITION
   STEP "BEA 1 Ebit1 Hand NOK [Camera Station]":   // S47, max time T#10S, warning time T#7S
              N    "GraDB2_FG02_Station_OP70".Workers.BEA[1].nok
   END_STEP
   TRANSITION "BEA 1 Ebit 1 Hand NOK ready [Camera Station]" FROM "BEA 1 Ebit1 Hand NOK [Camera Station]" TO "Controle Status [Camera Station]"   // T58, jump
      := "AlwaysTRUE";
   END_TRANSITION
   STEP "BEA 1 Ebit1 Repeat [Camera Station]":   // S48, max time T#10S, warning time T#7S
              N    "GraDB2_FG02_Station_OP70".Workers.BEA[1].repeat
   END_STEP
   TRANSITION "BEA 1 Ebit 1 Repeat active [Camera Station]" FROM "BEA 1 Ebit1 Repeat [Camera Station]" TO "Control BEA 1 Ebit 1 [Camera Station]"   // T59, jump
      := "AlwaysTRUE";
   END_TRANSITION
   STEP "Camera Process  [Camera Station]":   // S49, max time T#10S, warning time T#7S
      supervision V := NOT #"Proces Finished [Camera Station]".TT AND (#"Camera Process  [Camera Station]".U > t#1S);
              N    "GraDB2_FG02_Station_OP70".Camera.A.StartPRG[1]
              N    "GraDB2_FG02_Station_OP70".Camera.A.Start_active
   END_STEP
   TRANSITION "Proces Finished [Camera Station]" FROM "Camera Process  [Camera Station]" TO "Rate BEA1 Ebit 1 [Camera Station]"   // T60
      := "AnwDB_Omron_OP70_2".Output.Done AND "AnwDB_ProcessData_FG02_OP70".BEA[1].EBit[1].Finished AND "AnwDB_ProcessData_FG02_OP70".BEA[1].EBit[2].Finished AND "AnwDB_ProcessData_FG02_OP70".BEA[1].EBit[3].Finished AND "AnwDB_ProcessData_FG02_OP70".BEA[1].EBit[4].Finished AND "AnwDB_ProcessData_FG02_OP70".BEA[1].EBit[5].Finished AND "AnwDB_ProcessData_FG02_OP70".BEA[1].EBit[6].Finished AND "AnwDB_ProcessData_FG02_OP70".BEA[1].EBit[7].Finished AND "AnwDB_ProcessData_FG02_OP70".BEA[1].EBit[8].Finished;
   END_TRANSITION
   STEP "Restart Camera  [Camera Station]":   // S59, max time T#10S, warning time T#7S
      supervision V := NOT #"Camera Ready for Proces [Camera Station]".TT AND (#"Restart Camera  [Camera Station]".U > t#1S);
              N    "GraDB2_FG02_Station_OP70".Camera.A.Reset_outputs
   END_STEP
   TRANSITION "Camera Ready for Proces [Camera Station]" FROM "Restart Camera  [Camera Station]" TO "Camera delay"   // T74
      := "AnwDB_Omron_OP70_2".Output.Ready AND NOT "AnwDB_Omron_OP70_2".Output.Busy AND NOT "AnwDB_Omron_OP70_2".Output.Done;
   END_TRANSITION
   STEP "Camera delay":   // S63, max time T#10S, warning time T#7S
      supervision V := NOT #"Camera Ready for Proces [Camera Station]_1".TT AND (#"Camera delay".U > t#1S);
              N    "GraDB2_FG02_Station_OP70".Camera.A.Reset_outputs
   END_STEP
   TRANSITION "Camera Ready for Proces [Camera Station]_1" FROM "Camera delay" TO "Camera Process  [Camera Station]"   // T79
      := #"Camera delay".T > t#200MS;
   END_TRANSITION

   // permanent post-instructions
   NETWORK 1
   TITLE = Move interlocks from Ext block to ManualGraphControl DB
      "LTLL_ManualGraphInterlock"(ManualGraphExtOutput := #extBlock.output,
                              ManualGraphControlScreen := "LTLL_ManualGraphControl_OP70".screen[0]);
   NETWORK 2
   TITLE = Report step error
      "SysFC_NumOfSQErrors"(FLT := #RT_DATA.SQ_FLAGS.ERR_FLT,
                            Fault_SQ := "AnwDB_OperatingModes_OP70".BA[0].error_report_SK,
                            NumOf_Fault_SQ := "AnwDB_ZP_Alarm_OP70".FaultsNoSK_ST1);
   NETWORK 3
   TITLE = Basic position Step chain
      "GraDB2_FG02_Station_OP70".Home_SQ := (#INIT.X OR #"Waiting For pallet".X OR #"Finish SQ".X) AND (#"INIT [Camera Station]".X OR #"Waiting For Pallet [Camera Station]".X OR #"Finish SQ [Camera Station]".X);
END_FUNCTION_BLOCK
